// TwinCAT 3 PLC project Practice_V1
// ProgramVersion: 3.1.4024.0
// libraries:
//   Tc2_Standard, * (Beckhoff Automation GmbH)
//   Tc2_System, * (Beckhoff Automation GmbH)
//   Tc3_Module, * (Beckhoff Automation GmbH)
// project tree:
//   / PlcTask.TcTTO
//   POUs/ FB_Animal.TcPOU, FB_Dog.TcPOU, MAIN.TcPOU (not stored)
// real-time tasks:
//   TASK PlcTask: cycle T#10ms, priority 20, ADS port 350
//   TASK PlcTask1: cycle T#10ms, priority 21, ADS port 351
//   TASK PlcTask2: cycle T#10ms, priority 22, ADS port 352
//   TASK PlcTask3: cycle T#10ms, priority 23, ADS port 353

CONFIGURATION Practice_V1
    RESOURCE PLC ON TwinCAT3
        TASK PlcTask(INTERVAL := T#10ms, PRIORITY := 20);
        PROGRAM MAIN WITH PlcTask : MAIN;
    END_RESOURCE
END_CONFIGURATION

// ---- POUs/FB_Animal.TcPOU
FUNCTION_BLOCK FB_Animal
VAR
	 sOutput : STRING := '';
	 
	  x : INT := 8;
END_VAR

METHOD M_Eat
VAR_INPUT
END_VAR
THIS^.sOutput := 'Animal eats food';
END_METHOD

METHOD M_Sleep : BOOL
VAR_INPUT
END_VAR
THIS^.sOutput := 'Animal sleeps';
END_METHOD

END_FUNCTION_BLOCK

// ---- POUs/FB_Dog.TcPOU
FUNCTION_BLOCK FB_Dog EXTENDS FB_Animal

VAR
	 y : INT:=76;
END_VAR

x := 876;

METHOD M_Bark
VAR_INPUT
END_VAR
THIS^.sOutput := 'Dog barks';
END_METHOD

END_FUNCTION_BLOCK
